(* IEC 61131-3 sources: eCockpitGit/test_project/src/%F%00 Library/%F%Common Functions/%F%Module Value Conversion/%F%Real, 4 files *)

(* ---- %POU%FU_moduleValue3Point_As2Point_FromReal.st ---- *)
//Performs the conversion of a module value to a 3 point calibrated value
// |**Version**|**Author**| **Date** |**Changes**
// | 1         | NSN      | 29-03-22 | Creation
FUNCTION FU_moduleValue3Point_As2Point_FromReal : BOOL
VAR_INPUT
	value			:REAL;		//Value to convert value
	inMin			:REAL;		//Minimum value of calibration (point 1)
	inMax			:REAL;		//Maximum value of calibration (point 3)
END_VAR
VAR_IN_OUT
	data			:SModuleValueConversion3Point;	//3 Point conversion struct
END_VAR
VAR
	module			:AModule;
	valueType		:EValueType;
END_VAR

(*%!%__DELIMITER__%!%*)
module									:=		GMod.modMan.getModuleByUID(modUID:=data.moduleUID);
IF module <> 0 THEN
	CASE module^.SYS_valueType OF
		EValueType.digital:
			module^.SYS_valueDigital	:=		value <> inMin;
		EValueType.float32:
			module^.SYS_valueFloat32	:=		FU_rLinear2(XIn:=value,X1:=inMin,X2:=inMax,Y1:=data.midValue.float32,Y2:=data.maxValue.float32);
		EValueType.signed32,EValueType.enum:
			module^.SYS_valueSigned32	:=		TO_DINT(FU_rLinear2(XIn:=value,X1:=inMin,X2:=inMax,Y1:=data.midValue.float32,Y2:=data.maxValue.float32));
		EValueType.signed64:
			module^.SYS_valueSigned64	:=		TO_LINT(FU_rLinear2(XIn:=value,X1:=inMin,X2:=inMax,Y1:=data.midValue.float32,Y2:=data.maxValue.float32));
		EValueType.unsigned32:
			module^.SYS_valueUnsigned32	:=		TO_DWORD(FU_rLinear2(XIn:=value,X1:=inMin,X2:=inMax,Y1:=data.midValue.float32,Y2:=data.maxValue.float32));
		EValueType.unsigned64:
			module^.SYS_valueUnsigned64	:=		TO_LWORD(FU_rLinear2(XIn:=value,X1:=inMin,X2:=inMax,Y1:=data.midValue.float32,Y2:=data.maxValue.float32));
	END_CASE
END_IF

(* ---- %POU%FU_moduleValue3Point_As2Point_ToReal.st ---- *)
//Performs the conversion of a module value to a 3 point calibrated value
//Returns if the value is valid and the converted value
// |**Version**|**Author**| **Date** |**Changes**
// | 1         | NSN      | 29-03-22 | Creation
FUNCTION FU_moduleValue3Point_As2Point_ToReal : EValueValidity
VAR_OUTPUT
	value			:REAL;		//Converted value
END_VAR
VAR_INPUT
	outMin			:REAL;		//Minimum value of calibration (point 1)
	outMax			:REAL;		//Maximum value of calibration (point 3)
END_VAR
VAR_IN_OUT
	data			:SModuleValueConversion3Point;	//3 Point conversion struct
END_VAR
VAR
	module			:AModule;
	valueType		:EValueType;
END_VAR

(*%!%__DELIMITER__%!%*)
module									:=		GMod.modMan.getModuleByUID(modUID:=data.moduleUID);
IF module <> 0 THEN
	FU_moduleValue3Point_As2Point_ToReal:=		module^.SYS_isValid;
	IF FU_moduleValue3Point_As2Point_ToReal = EValueValidity.valid THEN
		CASE module^.SYS_valueType OF
			EValueType.digital:
				IF module^.SYS_valueDigital THEN
					value				:=		outMax;
				ELSE
					value				:=		outMin;
				END_IF
			EValueType.float32:
				value					:=		FU_rLinear2(XIn:=module^.SYS_valueFloat32,X1:=data.midValue.float32,X2:=data.maxValue.float32,Y1:=outMin,Y2:=outMax);
			EValueType.signed32,EValueType.enum:
				value					:=		FU_rLinear2(XIn:=TO_REAL(module^.SYS_valueSigned32),X1:=data.midValue.float32,X2:=data.maxValue.float32,Y1:=outMin,Y2:=outMax);
			EValueType.signed64:
				value					:=		FU_rLinear2(XIn:=TO_REAL(module^.SYS_valueSigned64),X1:=data.midValue.float32,X2:=data.maxValue.float32,Y1:=outMin,Y2:=outMax);
			EValueType.unsigned32:
				value					:=		FU_rLinear2(XIn:=TO_REAL(module^.SYS_valueUnsigned32),X1:=data.midValue.float32,X2:=data.maxValue.float32,Y1:=outMin,Y2:=outMax);
			EValueType.unsigned64:
				value					:=		FU_rLinear2(XIn:=TO_REAL(module^.SYS_valueUnsigned64),X1:=data.midValue.float32,X2:=data.maxValue.float32,Y1:=outMin,Y2:=outMax);
		END_CASE
	END_IF
ELSE
	FU_moduleValue3Point_As2Point_ToReal:=		EValueValidity.sourceInvalid;
END_IF

(* ---- %POU%FU_moduleValue3PointFromReal.st ---- *)
//Performs the conversion of a module value to a 3 point calibrated value
// |**Version**|**Author**| **Date** |**Changes**
// | 1         | NSN      | 29-03-22 | Creation
FUNCTION FU_moduleValue3PointFromReal : BOOL
VAR_INPUT
	value			:REAL;		//Value to convert value
	inMin			:REAL;		//Minimum value of calibration (point 1)
	inMid			:REAL;		//Middle value of calibration (point 2)
	inMax			:REAL;		//Maximum value of calibration (point 3)
END_VAR
VAR_IN_OUT
	data			:SModuleValueConversion3Point;	//3 Point conversion struct
END_VAR
VAR
	module			:AModule;
	valueType		:EValueType;
END_VAR

(*%!%__DELIMITER__%!%*)
module									:=		GMod.modMan.getModuleByUID(modUID:=data.moduleUID);
IF module <> 0 THEN
	CASE module^.SYS_valueType OF
		EValueType.digital:
			module^.SYS_valueDigital	:=		value <> inMid;
		EValueType.float32:
			module^.SYS_valueFloat32	:=		FU_rLinear3(XIn:=value,X1:=inMin,X2:=inMid,X3:=inMax,Y1:=data.minValue.float32,Y2:=data.midValue.float32,Y3:=data.maxValue.float32);
		EValueType.signed32,EValueType.enum:
			module^.SYS_valueSigned32	:=		TO_DINT(FU_rLinear3(XIn:=value,X1:=inMin,X2:=inMid,X3:=inMax,Y1:=data.minValue.float32,Y2:=data.midValue.float32,Y3:=data.maxValue.float32));
		EValueType.signed64:
			module^.SYS_valueSigned64	:=		TO_LINT(FU_rLinear3(XIn:=value,X1:=inMin,X2:=inMid,X3:=inMax,Y1:=data.minValue.float32,Y2:=data.midValue.float32,Y3:=data.maxValue.float32));
		EValueType.unsigned32:
			module^.SYS_valueUnsigned32	:=		TO_DWORD(FU_rLinear3(XIn:=value,X1:=inMin,X2:=inMid,X3:=inMax,Y1:=data.minValue.float32,Y2:=data.midValue.float32,Y3:=data.maxValue.float32));
		EValueType.unsigned64:
			module^.SYS_valueUnsigned64	:=		TO_LWORD(FU_rLinear3(XIn:=value,X1:=inMin,X2:=inMid,X3:=inMax,Y1:=data.minValue.float32,Y2:=data.midValue.float32,Y3:=data.maxValue.float32));
	END_CASE
END_IF

(* ---- %POU%FU_moduleValue3PointToReal.st ---- *)
//Performs the conversion of a module value to a 3 point calibrated value
//Returns if the value is valid and the converted value
// |**Version**|**Author**| **Date** |**Changes**
// | 1         | NSN      | 29-03-22 | Creation
FUNCTION FU_moduleValue3PointToReal : EValueValidity
VAR_OUTPUT
	value			:REAL;		//Converted value
END_VAR
VAR_INPUT
	outMin			:REAL;		//Minimum value of calibration (point 1)
	outMid			:REAL;		//Middle value of calibration (point 2)
	outMax			:REAL;		//Maximum value of calibration (point 3)
END_VAR
VAR_IN_OUT
	data			:SModuleValueConversion3Point;	//3 Point conversion struct
END_VAR
VAR
	module			:AModule;
	valueType		:EValueType;
END_VAR

(*%!%__DELIMITER__%!%*)
module									:=		GMod.modMan.getModuleByUID(modUID:=data.moduleUID);
IF module <> 0 THEN
	FU_moduleValue3PointToReal			:=		module^.SYS_isValid;
	IF FU_moduleValue3PointToReal = EValueValidity.valid THEN
		CASE module^.SYS_valueType OF
			EValueType.digital:
				IF module^.SYS_valueDigital THEN
					value				:=		outMax;
				ELSE
					value				:=		outMid;
				END_IF
			EValueType.float32:
				value					:=		FU_rLinear3(XIn:=module^.SYS_valueFloat32,X1:=data.minValue.float32,X2:=data.midValue.float32,X3:=data.maxValue.float32,Y1:=outMin,Y2:=outMid,Y3:=outMax);
			EValueType.signed32,EValueType.enum:
				value					:=		FU_rLinear3(XIn:=TO_REAL(module^.SYS_valueSigned32),X1:=data.minValue.float32,X2:=data.midValue.float32,X3:=data.maxValue.float32,Y1:=outMin,Y2:=outMid,Y3:=outMax);
			EValueType.signed64:
				value					:=		FU_rLinear3(XIn:=TO_REAL(module^.SYS_valueSigned64),X1:=data.minValue.float32,X2:=data.midValue.float32,X3:=data.maxValue.float32,Y1:=outMin,Y2:=outMid,Y3:=outMax);
			EValueType.unsigned32:
				value					:=		FU_rLinear3(XIn:=TO_REAL(module^.SYS_valueUnsigned32),X1:=data.minValue.float32,X2:=data.midValue.float32,X3:=data.maxValue.float32,Y1:=outMin,Y2:=outMid,Y3:=outMax);
			EValueType.unsigned64:
				value					:=		FU_rLinear3(XIn:=TO_REAL(module^.SYS_valueUnsigned64),X1:=data.minValue.float32,X2:=data.midValue.float32,X3:=data.maxValue.float32,Y1:=outMin,Y2:=outMid,Y3:=outMax);
		END_CASE
	END_IF
ELSE
	FU_moduleValue3PointToReal			:=		EValueValidity.sourceInvalid;
END_IF
